FUNCTION FB_SPS_zu_Nativ_INPUT_VAR : INPUT_VAR
VAR_INPUT
	INPUT: INPUT_VAR;
	
END_VAR
VAR
END_VAR

//Lineare Umrechnung der Eingangsgröße vom Typ INT in den nativen Wert vom Typ REAL
INPUT.REAL_VAR := INPUT.REAL_PARA_M * INPUT.INT_VAR_Input + INPUT.REAL_PARA_C;

//Übergabe an den Rückgabewert
FB_SPS_zu_Nativ_INPUT_VAR:=INPUT;

END_FUNCTION

(* stored: Version 1.1.0.1, ProductVersion 3.1.4019.2
   POU FB_SPS_zu_Nativ_INPUT_VAR: Id {f02bbc43-2c49-4ffe-9222-f75ffc30ebba}, SpecialFunc None *)
